{attribute addProperty BoxType "EP9128-0021-0017"}
{attribute addProperty Id "A_0010_EP9128_0021_0018A_0010_EP9128_0021_0018_A4E842674566570.75A_0007_EP9128_0021_0017_2_EP9128_1021EP9128_179A0949162A_0007_EP9128_0021_0017_3_EP9128_2021EP9128_179A0949162"}
{attribute addProperty CRC "177452393"}
{attribute addProperty SizeInBites "4598"}
{attribute addProperty SizeInBytes "574.75"}
TYPE A_0007_EP9128_0021_0017_0A93B569 EXTENDS EP9128_179A0949 :
STRUCT
	{attribute addProperty Name "A_0010_EP9128_0021_0018"}
	A_0010_EP9128_0021_0018 : A_0010_EP9128_0021_0018_A4E84267;
	{attribute addProperty Name "A_0007_EP9128_0021_0017_2_EP9128_1021"}
	A_0007_EP9128_0021_0017_2_EP9128_1021 : EP9128_179A0949;
	{attribute addProperty Name "A_0007_EP9128_0021_0017_3_EP9128_2021"}
	A_0007_EP9128_0021_0017_3_EP9128_2021 : EP9128_179A0949;
END_STRUCT
END_TYPE

(* stored: Version 1.2.0.0, ProductVersion 3.1.4024.9
   DUT A_0007_EP9128_0021_0017_0A93B569: Id {75f46232-eb02-4f8f-a918-70fba028c05c} *)
